// TIA Portal project "test项目" (V20)

(* hardware
DEVICE "S7-1200 station_1"  S7-1200 Station
   slot 0: "Rack_0"  S7-1200 Rack  Rack  V1.0
   slot 1: "PLC_1"  CPU 1215C DC/DC/DC  6ES7 215-1AG40-0XB0  V4.6
   slot 3: "CB 1241 (RS485)"  CB 1241 (RS485)  6ES7 241-1CH30-1XB0  V1.0
*)

// ===== PLC "PLC_1"  CPU 1215C DC/DC/DC =====

VAR_GLOBAL   // PLC tag table "默认变量表"
   "System_Byte" AT %MB1 : Byte;
   "FirstScan" AT %M1.0 : Bool;
   "DiagStatusUpdate" AT %M1.1 : Bool;
   "AlwaysTRUE" AT %M1.2 : Bool;
   "AlwaysFALSE" AT %M1.3 : Bool;
   "Clock_Byte" AT %MB0 : Byte;
   "Clock_10Hz" AT %M0.0 : Bool;
   "Clock_5Hz" AT %M0.1 : Bool;
   "Clock_2.5Hz" AT %M0.2 : Bool;
   "Clock_2Hz" AT %M0.3 : Bool;
   "Clock_1.25Hz" AT %M0.4 : Bool;
   "Clock_1Hz" AT %M0.5 : Bool;
   "Clock_0.625Hz" AT %M0.6 : Bool;
   "Clock_0.5Hz" AT %M0.7 : Bool;
   "Tag_1" AT %Q0.6 : Bool;
   "Tag_2" AT %I0.3 : Bool;
   "Tag_3" AT %I0.4 : Bool;
   "Tag_4" AT %I0.5 : Bool;
   "Tag_5" AT %I0.6 : Bool;
   "Tag_6" AT %I0.7 : Bool;
   "Tag_7" AT %M2.4 : Bool;
   "Tag_8" AT %M2.5 : Bool;
   "Tag_9" AT %M2.3 : Bool;
   "Tag_10" AT %QB0 : Byte;
END_VAR

VAR_GLOBAL   // PLC tag table "input"
   "limit_left" AT %I0.0 : Bool;
   "zero_point" AT %I0.1 : Bool;
   "limit_right" AT %I0.2 : Bool;
   "start" AT %I0.0 : Bool;
   "reset" AT %I0.1 : Bool;
   "b_a" AT %I0.2 : Bool;
   "b_b" AT %I0.3 : Bool;
   "b_c" AT %I0.4 : Bool;
   "b_d" AT %I0.5 : Bool;
END_VAR

VAR_GLOBAL   // PLC tag table "output"
   "puls_plus" AT %Q0.0 : Bool;
   "red_w" AT %Q0.1 : Bool;
   "dir_plus" AT %Q0.2 : Bool;
   "light_a" AT %Q0.3 : Bool;
   "light_b" AT %Q0.4 : Bool;
   "light_c" AT %Q0.5 : Bool;
   "light_d" AT %Q0.6 : Bool;
   "light_answer" AT %Q0.7 : Bool;
   "sound_answer" AT %Q1.2 : Bool;
END_VAR

VAR_GLOBAL   // PLC tag table "intermedia"
   "p1" AT %M2.0 : Bool;
   "p2" AT %M2.1 : Bool;
END_VAR

DATA_BLOCK "抢答器FB_SCL_DB"   // DB6
{ S7_Optimized_Access := 'TRUE' }
VERSION : 0.1
// stored: InstanceOfName 抢答器FB_SCL
"抢答器FB_SCL"
BEGIN
END_DATA_BLOCK

// folder: 作业

DATA_BLOCK "喷泉LAD数据块"   // DB1
{ S7_Optimized_Access := 'TRUE' }
VERSION : 0.1
   VAR
      started : Bool;
      stopped : Bool;
      running : Bool;
      cache : Array[0..10] of Bool;
      step1 : USInt;
      step2 : USInt;
      Static_1 : USInt;
      timer1 : IEC_TIMER;
      timer2 : IEC_TIMER;
      timer3 : IEC_TIMER;
      timer4 : IEC_TIMER;
      timer5 : IEC_TIMER;
      timer6 : IEC_TIMER;
      timer7 : IEC_TIMER;
      timer8 : IEC_TIMER;
      timer9 : IEC_TIMER;
      timer10 : IEC_TIMER;
      pt_1 : Time;
      pt_2 : Time;
   END_VAR
BEGIN
END_DATA_BLOCK

DATA_BLOCK "交通红绿灯_流程SCL_DB"   // DB2
{ S7_Optimized_Access := 'TRUE' }
VERSION : 0.1
// stored: InstanceOfName 交通红绿灯_流程SCL
"交通红绿灯_流程SCL"
BEGIN
END_DATA_BLOCK

DATA_BLOCK "交通红绿灯_比较SCL_DB"   // DB3
{ S7_Optimized_Access := 'TRUE' }
VERSION : 0.1
// stored: InstanceOfName 交通红绿灯_比较SCL
"交通红绿灯_比较SCL"
BEGIN
END_DATA_BLOCK

DATA_BLOCK "喷泉_DB"   // DB4
{ S7_Optimized_Access := 'TRUE' }
VERSION : 0.1
// stored: InstanceOfName 喷泉
"喷泉"
BEGIN
END_DATA_BLOCK

DATA_BLOCK "抢答器LAD数据块_1"   // DB5
{ S7_Optimized_Access := 'TRUE' }
VERSION : 0.1
   VAR
      started : Bool;
      success : Bool;
      success_a : Bool;
      success_b : Bool;
      success_c : Bool;
      success_d : Bool;
      cache : Array[0..10] of Bool;
      timer1 : IEC_TIMER;
      timer2 : IEC_TIMER;
      timer3 : IEC_TIMER;
      timer8 : IEC_TIMER;
      timer9 : IEC_TIMER;
      timer7 : IEC_TIMER;
      timer6 : IEC_TIMER;
      timer5 : IEC_TIMER;
      timer4 : IEC_TIMER;
      eligible_a : Bool;
      eligible_b : Bool;
      eligible_c : Bool;
      eligible_d : Bool;
      cnt : SInt;
   END_VAR
BEGIN
END_DATA_BLOCK

// folder: (top level)

FUNCTION_BLOCK "抢答器FB_SCL"   // FB4, SCL
{ S7_Optimized_Access := 'TRUE' }
VERSION : 0.1
   VAR
      started : Bool;
      start_TRIG_Instance : R_TRIG;
      reset_TRIG_Instance : R_TRIG;
      b_a_TRIG_Instance : R_TRIG;
      b_b_TRIG_Instance : R_TRIG;
      b_c_TRIG_Instance : R_TRIG;
      b_d_TRIG_Instance : R_TRIG;
      success_a : Bool;
      success_b : Bool;
      success_c : Bool;
      success_d : Bool;
      eligible_a : Bool;
      eligible_b : Bool;
      eligible_c : Bool;
      eligible_d : Bool;
      timer1 : IEC_TIMER;
      timer2 : IEC_TIMER;
      IEC_Timer_0_Instance : TON_TIME;
      IEC_Timer_0_Instance_1 : TON_TIME;
      IEC_Timer_0_Instance_2 : TON_TIME;
      pt_1 : Time;
      pt_2 : Time;
      pt_3 : Time;
      cnt : SInt;
   END_VAR
BEGIN
   If "FirstScan" THEN
       #started := 0;
   END_IF;

   #start_TRIG_Instance(CLK := "start");
   #reset_TRIG_Instance(CLK := "reset");
   #b_a_TRIG_Instance(CLK := "b_a");
   #b_b_TRIG_Instance(CLK := "b_b");
   #b_c_TRIG_Instance(CLK := "b_c");
   #b_d_TRIG_Instance(CLK := "b_d");
   #pt_1 := t#3s;
   #pt_2 := #pt_3 := t#1s;
   #IEC_Timer_0_Instance(IN := #started,
                         PT := #pt_1);

   #IEC_Timer_0_Instance_1(IN := #IEC_Timer_0_Instance.Q,
                           PT := #pt_2);

   #IEC_Timer_0_Instance_2(IN := #IEC_Timer_0_Instance_1.Q,
                           PT := #pt_3);

   If #start_TRIG_Instance.Q AND NOT #started THEN
       #started := #eligible_a := #eligible_b := #eligible_c := #eligible_d := 1;
       #success_a := #success_b := #success_c := #success_d := 0;
       #cnt := 0;

   END_IF;

   If #reset_TRIG_Instance.Q THEN
       #started := 0;
       "light_a" := "light_b" := "light_c" := "light_d" := "light_answer" := "sound_answer" := 0;
   END_IF;

   If #started THEN
       If NOT #IEC_Timer_0_Instance.Q THEN
           "light_a" := #eligible_a;
           "light_b" := #eligible_b;
           "light_c" := #eligible_c;
           "light_d" := #eligible_d;
           "light_answer" := "sound_answer" := 1;
           If #b_a_TRIG_Instance.Q THEN
               #eligible_a := 0;
           END_IF;
           If #b_b_TRIG_Instance.Q THEN
               #eligible_b := 0;
           END_IF;
           If #b_c_TRIG_Instance.Q THEN
               #eligible_c := 0;
           END_IF;
           If #b_d_TRIG_Instance.Q THEN
               #eligible_d := 0;
           END_IF;
       END_IF;

       If #IEC_Timer_0_Instance.Q THEN
           "light_a" := "light_b" := "light_c" := "light_d" := 0;
           If #eligible_a AND #b_a_TRIG_Instance.Q THEN
               #eligible_b := 0;
               #eligible_c := 0;
               #eligible_d := 0;
               #eligible_a := 0;
               #success_a := 1;
               RESET_TIMER(#IEC_Timer_0_Instance_1);
           END_IF;
           If #eligible_b AND #b_b_TRIG_Instance.Q THEN
               #eligible_b := 0;
               #eligible_c := 0;
               #eligible_d := 0;
               #eligible_a := 0;
               #success_b := 1;
               RESET_TIMER(#IEC_Timer_0_Instance_1);
           END_IF;
           If #eligible_c AND #b_c_TRIG_Instance.Q THEN
               #eligible_b := 0;
               #eligible_c := 0;
               #eligible_d := 0;
               #eligible_a := 0;
               #success_c := 1;
               RESET_TIMER(#IEC_Timer_0_Instance_1);
           END_IF;
           If #eligible_d AND #b_d_TRIG_Instance.Q THEN
               #eligible_b := 0;
               #eligible_c := 0;
               #eligible_d := 0;
               #eligible_a := 0;
               #success_d := 1;
               RESET_TIMER(#IEC_Timer_0_Instance_1);
           END_IF;

           If #success_a THEN
               "light_a" := NOT #IEC_Timer_0_Instance_1.Q OR #cnt = 3;
               If #IEC_Timer_0_Instance_2.Q THEN
                   RESET_TIMER(#IEC_Timer_0_Instance_1);
                   #cnt += 1;
               END_IF;
               If #cnt = 3 THEN
                   RESET_TIMER(#IEC_Timer_0_Instance_1);
               END_IF;
           END_IF;
           If #success_b THEN
               "light_b" := NOT #IEC_Timer_0_Instance_1.Q OR #cnt = 3;
               If #IEC_Timer_0_Instance_2.Q THEN
                   RESET_TIMER(#IEC_Timer_0_Instance_1);
                   #cnt += 1;
               END_IF;
               If #cnt = 3 THEN
                   RESET_TIMER(#IEC_Timer_0_Instance_1);
               END_IF;
           END_IF;
           If #success_c THEN
               "light_c" := NOT #IEC_Timer_0_Instance_1.Q OR #cnt = 3;
               If #IEC_Timer_0_Instance_2.Q THEN
                   RESET_TIMER(#IEC_Timer_0_Instance_1);
                   #cnt += 1;
               END_IF;
               If #cnt = 3 THEN
                   RESET_TIMER(#IEC_Timer_0_Instance_1);
               END_IF;
           END_IF;
           If #success_d THEN
               "light_d" := NOT #IEC_Timer_0_Instance_1.Q OR #cnt = 3;
               If #IEC_Timer_0_Instance_2.Q THEN
                   RESET_TIMER(#IEC_Timer_0_Instance_1);
                   #cnt += 1;
               END_IF;
               If #cnt = 3 THEN
                   RESET_TIMER(#IEC_Timer_0_Instance_1);
               END_IF;
           END_IF;
       END_IF;
   END_IF;
END_FUNCTION_BLOCK

ORGANIZATION_BLOCK "Main"   // OB1, LAD, ProgramCycle
TITLE = "Main Program Sweep (Cycle)"
{ S7_Optimized_Access := 'TRUE' }
VERSION : 0.1
   VAR_INPUT
      Initial_Call : Bool;   // Initial call of this OB
      Remanence : Bool;   // =True, if remanent data are available
   END_VAR
BEGIN

REGION Network 1 (SCL)
   (*



   *)
END_REGION

REGION Network 2
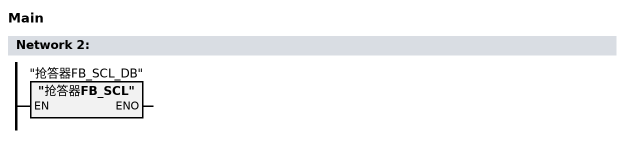
   RUNG wire#powerrail
      "抢答器FB_SCL_DB"()
   END_RUNG
   // the same network as SCL:
   "抢答器FB_SCL_DB"();   // "抢答器FB_SCL"
END_REGION
END_ORGANIZATION_BLOCK

// folder: 作业

FUNCTION_BLOCK "喷泉"   // FB1, SCL
{ S7_Optimized_Access := 'TRUE' }
VERSION : 0.1
   VAR
      timer1 : TON_TIME;
      timer2 : TON_TIME;
      pt_1 : Time;
      pt_2 : Time;
      step1 : USInt;
      step2 : USInt;
      step3 : USInt;
      started : Bool;
      stopped : Bool;
      running : Bool;
      R_TRIG_Instance : R_TRIG;
      R_TRIG_Instance_1 : R_TRIG;
      R_TRIG_Instance_2 : R_TRIG;
   END_VAR
BEGIN
   #timer1(IN := #running,
           PT := #pt_1);
   #timer2(IN := #timer1.Q,
           PT := #pt_2);
   #R_TRIG_Instance(CLK:="start");
   #R_TRIG_Instance_1(CLK:="reset");
   #R_TRIG_Instance_2(CLK:=#started);

   IF #R_TRIG_Instance.Q THEN
       #started := 1;
   END_IF;

   IF #R_TRIG_Instance_1.Q THEN
       #stopped := 1;
   END_IF;

   IF #R_TRIG_Instance_2.Q THEN
       #running := 1;
       #pt_1 := t#5s;
       #pt_2 := t#5s;
       RESET_TIMER(#timer1);
       #step1 := #step2 := #step3 := 0;
   END_IF;

   IF #running THEN
       IF #step1 = 0 THEN
           "light_a" := NOT #timer1.Q;
           "light_b" := NOT #timer2.Q AND #timer1.Q;
           IF #timer2.Q THEN
               #step1 += 1;
               RESET_TIMER(#timer1);
           END_IF;
       END_IF;

       IF #step1 = 1 THEN
           "light_a" := "light_b" := NOT #timer1.Q;
           IF #timer1.Q THEN
               #step1 += 1;
               #pt_1 := #pt_2 := t#1s;
               RESET_TIMER(#timer1);
           END_IF;
       END_IF;

       IF #step1 = 2 THEN
           "light_c" := NOT #timer1.Q;
           IF #timer2.Q THEN
               #step2 += 1;
               RESET_TIMER(#timer1);
           END_IF;
           IF #step2 = 5 THEN
               #step1 += 1;
               #pt_1 := t#5s;
               RESET_TIMER(#timer1);
               #step2 := 0;
           END_IF;
       END_IF;

       IF #step1 = 3 THEN
           "light_a" := "light_b" := NOT #timer1.Q;
           IF #timer1.Q THEN
               #step1 += 1;
               #pt_1 := t#2s;
               RESET_TIMER(#timer1);
           END_IF;
       END_IF;

       IF #step1 = 4 THEN
           CASE #step3 OF
               0:
                   "light_a" := NOT #timer1.Q;
               1:
                   "light_b" := NOT #timer1.Q;
               2:
                   "light_c" := NOT #timer1.Q;
           END_CASE;

           IF #timer1.Q THEN
               #step3 += 1;
               IF #step3 = 3 THEN
                   #step2 += 1;
                   #step3 := 0;
               END_IF;
               IF #step2 = 3 THEN
                   #step1 += 1;
                   #step2 := 0;
                   #pt_1 := t#5S;
               END_IF;
               RESET_TIMER(#timer1);
           END_IF;
       END_IF;

       IF #step1 = 5 THEN
           IF #timer1.Q THEN
               #running := NOT #stopped;
               #started := #running;
               #pt_1 := #pt_2 := t#5s;
               #step1 := #step2 := #step3 := 0;
               RESET_TIMER(#timer1);
           END_IF;
       END_IF;
   END_IF;
END_FUNCTION_BLOCK

FUNCTION_BLOCK "交通红绿灯_流程SCL"   // FB2, LAD
{ S7_Optimized_Access := 'TRUE' }
VERSION : 0.1
   VAR
      start_pressed_trig : R_TRIG;
      stop_pressed_trig : R_TRIG;
      start_trig : R_TRIG;
      started : Bool;
      stoped : Bool;
      step_w : Byte;
      step_s : Byte;
      Timer_0 : TON_TIME;
      Timer_1 : TON_TIME;
      Timer_2 : TON_TIME;
      Timer_3 : TON_TIME;
      time_w : Time;
      time_s : Time;
   END_VAR
BEGIN

REGION Network 2 (SCL)
   IF "FirstScan" THEN
       #started := #stoped := 0;
       #step_w := #step_s := 0;
   END_IF;

   //initiate
   #start_pressed_trig(CLK := "limit_left");
   #stop_pressed_trig(CLK := "zero_point");
   #start_trig(CLK := #started);

   #Timer_0(IN := #started, PT := #time_w);
   #Timer_1(IN := #started, PT := #time_s);
   #Timer_2(IN := "AlwaysTRUE", PT := t#500ms);
   #Timer_3(IN := #Timer_2.Q,PT := t#500ms);
   IF #Timer_3.Q THEN
       RESET_TIMER(#Timer_2);
   END_IF;

   IF #start_pressed_trig.Q THEN
       #started := 1;
       #stoped := 0;
   END_IF;

   IF #start_trig.Q THEN
       #stoped := 0;
       #step_s := #step_w := 0;
       "light_a" := "puls_plus" := "dir_plus" := "light_c" := "red_w" := "light_b" := 0;
       #time_w := t#5s;
       #time_s := t#10s;
       RESET_TIMER(#Timer_0);
       RESET_TIMER(#Timer_1);
   END_IF;

   IF #stop_pressed_trig.Q THEN
       #stoped := 1;
   END_IF;

   IF #started THEN
       //东西向
       IF #step_w = 0 THEN
           "puls_plus" := 1;
           IF #Timer_0.Q THEN
               "puls_plus" := 0;
               RESET_TIMER(#Timer_0);
               #time_w := T#3s;
               #step_w += 1;
           END_IF;
       END_IF;

       IF #step_w = 1 THEN
           "puls_plus" := #Timer_2.Q;
           IF #Timer_0.Q THEN
               "puls_plus" := 0;
               RESET_TIMER(#Timer_0);
               #time_w := T#2s;
               #step_w += 1;
           END_IF;
       END_IF;

       IF #step_w = 2 THEN
           "dir_plus" := 1;
           IF #Timer_0.Q THEN
               "dir_plus" := 0;
               RESET_TIMER(#Timer_0);
               #time_w := T#10s;
               #step_w += 1;
           END_IF;
       END_IF;

       IF #step_w = 3 THEN
           "red_w":= 1;
           IF #Timer_0.Q THEN
               "red_w" := 0;
               RESET_TIMER(#Timer_0);
               #time_w := T#5s;
               #step_w := 0;
           END_IF;
       END_IF;

       //南北向
       IF #step_s = 0 THEN
           "light_b" := 1;
           IF #Timer_1.Q THEN
               "light_b" := 0;
               RESET_TIMER(#Timer_1);
               #time_s := T#5s;
               #step_s += 1;
           END_IF;
       END_IF;

       IF #step_s = 1 THEN
           "light_a" := 1;
           IF #Timer_1.Q THEN
               "light_a" := 0;
               RESET_TIMER(#Timer_1);
               #time_s := T#3s;
               #step_s += 1;
           END_IF;
       END_IF;

       IF #step_s = 2 THEN
          "light_a" := #Timer_2.Q;
          IF #Timer_1.Q THEN
              "light_a" := 0;
               RESET_TIMER(#Timer_1);
               #time_s := T#2s;
               #step_s += 1;
           END_IF;
       END_IF;

       IF #step_s = 3 THEN
           "light_c" := 1;
           IF #Timer_1.Q THEN
               "light_c" := 0;
               RESET_TIMER(#Timer_1);
               #time_s := T#10s;
               #step_s := 0;
               #step_w := 0;
               "red_w" := 0;
               RESET_TIMER(#Timer_0);
               #time_w := T#5s;
               #step_w := 0;

               IF #stoped THEN
                   #started := 0;
                   #stoped := 0;
               END_IF;
           END_IF;
       END_IF;
   END_IF;

   IF NOT #stoped AND NOT #started THEN
       "light_c" := #Timer_2.Q;
       "dir_plus" := #Timer_2.Q;
   END_IF;
END_REGION
END_FUNCTION_BLOCK

FUNCTION_BLOCK "交通红绿灯_比较SCL"   // FB3, LAD
{ S7_Optimized_Access := 'TRUE' }
VERSION : 0.1
   VAR
      start_pressed_trig : R_TRIG;
      stop_pressed_trig : R_TRIG;
      start_trig : R_TRIG;
      started : Bool;
      stoped : Bool;
      step_w : Byte;
      step_s : Byte;
      Timer_0 : TON_TIME;
      Timer_1 : TON_TIME;
      Timer_2 : TON_TIME;
      Timer_3 : TON_TIME;
      time_w : Time;
      time_s : Time;
      button : Array[0..10] of Bool;
      b1 : Bool;
      b2 : Bool;
      b4 : Bool;
      b3 : Bool;
      b5 : Bool;
   END_VAR
BEGIN

REGION Network 2 (SCL)
   IF "FirstScan" THEN
       #started := #stoped := 0;
       #step_w := #step_s := 0;
   END_IF;

   //initiate
   #start_pressed_trig(CLK := "limit_left");
   #stop_pressed_trig(CLK := "zero_point");
   #start_trig(CLK := #started);

   #Timer_0(IN := #started, PT := t#20S);
   #Timer_2(IN := "AlwaysTRUE", PT := t#500ms);
   #Timer_3(IN := #Timer_2.Q,PT := t#500ms);
   IF #Timer_3.Q THEN
       RESET_TIMER(#Timer_2);
   END_IF;

   IF #start_pressed_trig.Q THEN
       #started := 1;
       #stoped := 0;
   END_IF;

   IF #start_trig.Q THEN
       #stoped := 0;
       RESET_TIMER(#Timer_0);
       RESET_TIMER(#Timer_2);
   END_IF;

   IF #stop_pressed_trig.Q THEN
       #stoped := 1;
   END_IF;

   IF #started THEN
       //东西向
       "puls_plus" := #Timer_0.ET > t#0s AND #Timer_0.ET <= t#5s OR (#Timer_0.ET > t#5s AND #Timer_0.ET <= t#8s AND #Timer_2.Q);
       "dir_plus" := #Timer_0.ET > t#8s AND #Timer_0.ET <= t#10s;
       "red_w" := #Timer_0.ET > t#10s AND #Timer_0.ET <= t#20s;

       //南北向
       "light_b" := #Timer_0.ET > t#0s AND #Timer_0.ET <= t#10s;
       "light_a" := #Timer_0.ET > t#10s AND #Timer_0.ET <= t#13s OR (#Timer_0.ET > t#13s AND #Timer_0.ET <= t#15s AND #Timer_2.Q);
       "light_c" := #Timer_0.ET > t#15s AND #Timer_0.ET < t#20s;

       IF #Timer_0.ET >= t#20S THEN
           RESET_TIMER(#Timer_0);
           RESET_TIMER(#Timer_1);

           #started := NOT #stoped;
           #stoped := 0;
       END_IF;
   END_IF;

   IF NOT #stoped AND NOT #started THEN
       "light_a" := "puls_plus" := "light_b" := "red_w" := 0;
       "light_c" := #Timer_2.Q;
       "dir_plus" := #Timer_2.Q;
   END_IF;
END_REGION
END_FUNCTION_BLOCK

FUNCTION "红绿灯_FC" : Void   // FC1, LAD
{ S7_Optimized_Access := 'TRUE' }
VERSION : 0.1
   VAR_TEMP   // added for the SCL form of the ladder/FBD networks
      _w1 : Bool;
      _w2 : Bool;
      _w3 : Bool;
   END_VAR
BEGIN

REGION Network 1
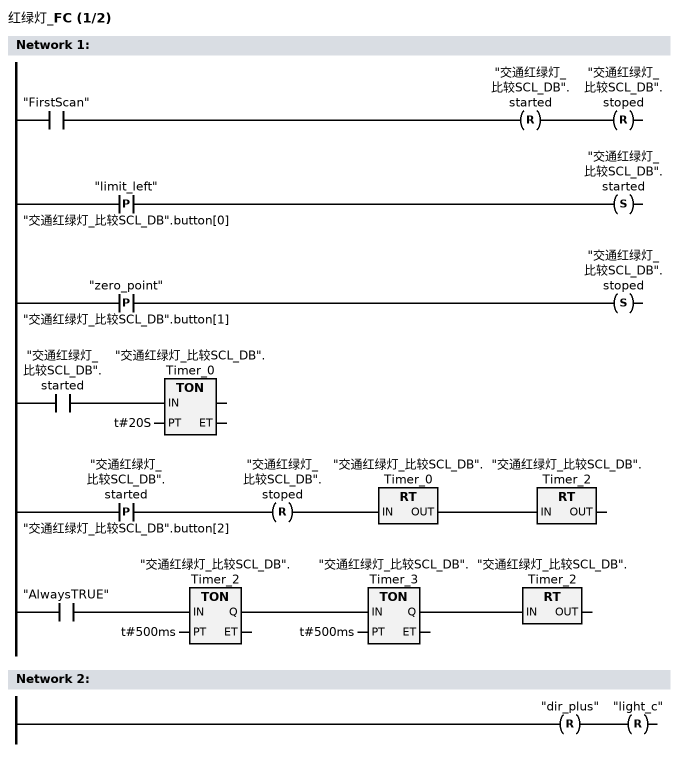
   IF "FirstScan" THEN
       "交通红绿灯_比较SCL_DB".started := FALSE;
       "交通红绿灯_比较SCL_DB".stoped := FALSE;
   END_IF;
   #_w1 := "limit_left" AND NOT "交通红绿灯_比较SCL_DB".button[0];   // rising edge of "limit_left"
   "交通红绿灯_比较SCL_DB".button[0] := "limit_left";
   IF #_w1 THEN "交通红绿灯_比较SCL_DB".started := TRUE; END_IF;
   #_w2 := "zero_point" AND NOT "交通红绿灯_比较SCL_DB".button[1];   // rising edge of "zero_point"
   "交通红绿灯_比较SCL_DB".button[1] := "zero_point";
   IF #_w2 THEN "交通红绿灯_比较SCL_DB".stoped := TRUE; END_IF;
   "交通红绿灯_比较SCL_DB".Timer_0.TON(IN := "交通红绿灯_比较SCL_DB".started, PT := t#20S);
   #_w3 := "交通红绿灯_比较SCL_DB".started AND NOT "交通红绿灯_比较SCL_DB".button[2];   // rising edge of "交通红绿灯_比较SCL_DB".started
   "交通红绿灯_比较SCL_DB".button[2] := "交通红绿灯_比较SCL_DB".started;
   IF #_w3 THEN
       "交通红绿灯_比较SCL_DB".stoped := FALSE;
       RESET_TIMER("交通红绿灯_比较SCL_DB".Timer_0);
       RESET_TIMER("交通红绿灯_比较SCL_DB".Timer_2);
   END_IF;
   "交通红绿灯_比较SCL_DB".Timer_2.TON(IN := "AlwaysTRUE", PT := t#500ms);
   "交通红绿灯_比较SCL_DB".Timer_3.TON(IN := "交通红绿灯_比较SCL_DB".Timer_2.Q, PT := t#500ms);
   IF "交通红绿灯_比较SCL_DB".Timer_3.Q THEN RESET_TIMER("交通红绿灯_比较SCL_DB".Timer_2); END_IF;
END_REGION

REGION Network 2
   RUNG wire#powerrail
      R_Coil( "dir_plus" )
      R_Coil( "light_c" )
   END_RUNG
   // the same network as SCL:
   "dir_plus" := FALSE;
   "light_c" := FALSE;
END_REGION

REGION Network 3
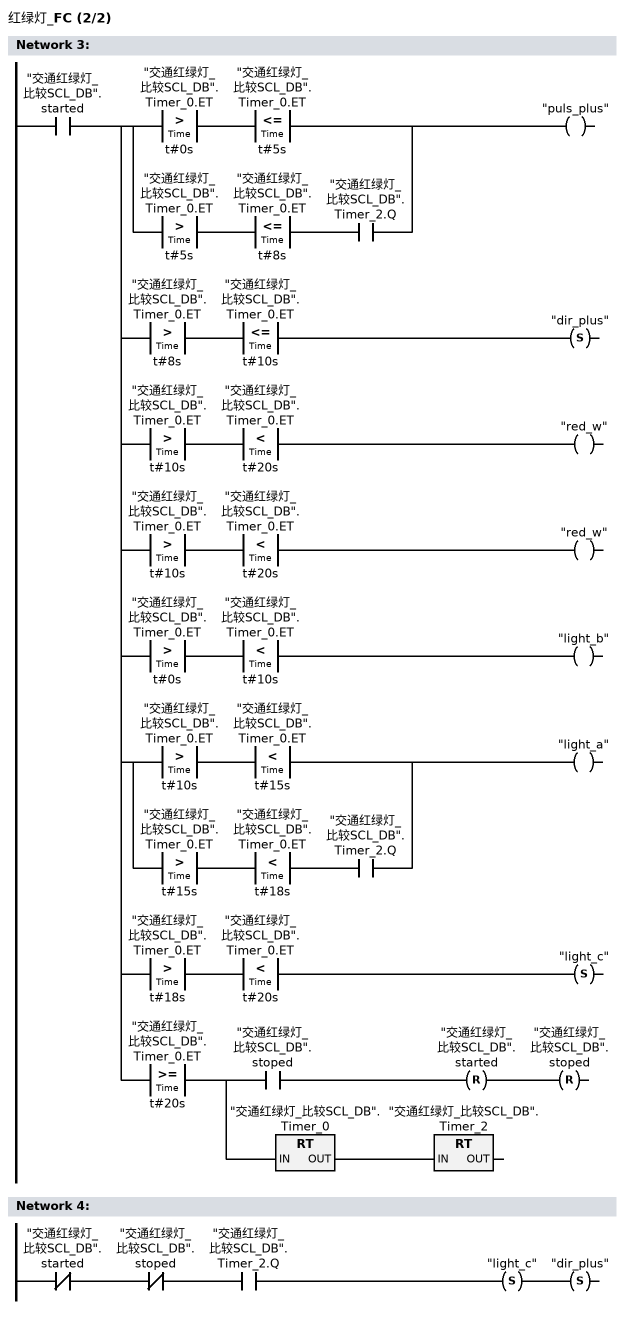
   RUNG wire#powerrail
      Contact( "交通红绿灯_比较SCL_DB".started )
      wire#w1
      { S7_Templates := "SrcType := Time" } GT_Contact(in1 := "交通红绿灯_比较SCL_DB".Timer_0.ET, in2 := t#0s)
      { S7_Templates := "SrcType := Time" } LE_Contact(in1 := "交通红绿灯_比较SCL_DB".Timer_0.ET, in2 := t#5s)
      wire#w2
      Coil( "puls_plus" )
   END_RUNG
   RUNG wire#w1
      { S7_Templates := "SrcType := Time" } GT_Contact(in1 := "交通红绿灯_比较SCL_DB".Timer_0.ET, in2 := t#5s)
      { S7_Templates := "SrcType := Time" } LE_Contact(in1 := "交通红绿灯_比较SCL_DB".Timer_0.ET, in2 := t#8s)
      Contact( "交通红绿灯_比较SCL_DB".Timer_2.Q )
   END_RUNG wire#w2
   RUNG wire#w1
      { S7_Templates := "SrcType := Time" } GT_Contact(in1 := "交通红绿灯_比较SCL_DB".Timer_0.ET, in2 := t#8s)
      { S7_Templates := "SrcType := Time" } LE_Contact(in1 := "交通红绿灯_比较SCL_DB".Timer_0.ET, in2 := t#10s)
      S_Coil( "dir_plus" )
   END_RUNG
   RUNG wire#w1
      { S7_Templates := "SrcType := Time" } GT_Contact(in1 := "交通红绿灯_比较SCL_DB".Timer_0.ET, in2 := t#10s)
      { S7_Templates := "SrcType := Time" } LT_Contact(in1 := "交通红绿灯_比较SCL_DB".Timer_0.ET, in2 := t#20s)
      Coil( "red_w" )
   END_RUNG
   RUNG wire#w1
      { S7_Templates := "SrcType := Time" } GT_Contact(in1 := "交通红绿灯_比较SCL_DB".Timer_0.ET, in2 := t#10s)
      { S7_Templates := "SrcType := Time" } LT_Contact(in1 := "交通红绿灯_比较SCL_DB".Timer_0.ET, in2 := t#20s)
      Coil( "red_w" )
   END_RUNG
   RUNG wire#w1
      { S7_Templates := "SrcType := Time" } GT_Contact(in1 := "交通红绿灯_比较SCL_DB".Timer_0.ET, in2 := t#0s)
      { S7_Templates := "SrcType := Time" } LT_Contact(in1 := "交通红绿灯_比较SCL_DB".Timer_0.ET, in2 := t#10s)
      Coil( "light_b" )
   END_RUNG
   RUNG wire#w1
      { S7_Templates := "SrcType := Time" } GT_Contact(in1 := "交通红绿灯_比较SCL_DB".Timer_0.ET, in2 := t#10s)
      { S7_Templates := "SrcType := Time" } LT_Contact(in1 := "交通红绿灯_比较SCL_DB".Timer_0.ET, in2 := t#15s)
      wire#w3
      Coil( "light_a" )
   END_RUNG
   RUNG wire#w1
      { S7_Templates := "SrcType := Time" } GT_Contact(in1 := "交通红绿灯_比较SCL_DB".Timer_0.ET, in2 := t#15s)
      { S7_Templates := "SrcType := Time" } LT_Contact(in1 := "交通红绿灯_比较SCL_DB".Timer_0.ET, in2 := t#18s)
      Contact( "交通红绿灯_比较SCL_DB".Timer_2.Q )
   END_RUNG wire#w3
   RUNG wire#w1
      { S7_Templates := "SrcType := Time" } GT_Contact(in1 := "交通红绿灯_比较SCL_DB".Timer_0.ET, in2 := t#18s)
      { S7_Templates := "SrcType := Time" } LT_Contact(in1 := "交通红绿灯_比较SCL_DB".Timer_0.ET, in2 := t#20s)
      S_Coil( "light_c" )
   END_RUNG
   RUNG wire#w1
      { S7_Templates := "SrcType := Time" } GE_Contact(in1 := "交通红绿灯_比较SCL_DB".Timer_0.ET, in2 := t#20s)
      wire#w4
      Contact( "交通红绿灯_比较SCL_DB".stoped )
      R_Coil( "交通红绿灯_比较SCL_DB".started )
      R_Coil( "交通红绿灯_比较SCL_DB".stoped )
   END_RUNG
   RUNG wire#w4
      RT_Coil( "交通红绿灯_比较SCL_DB".Timer_0 )
      RT_Coil( "交通红绿灯_比较SCL_DB".Timer_2 )
   END_RUNG
   // the same network as SCL:
   "puls_plus" := "交通红绿灯_比较SCL_DB".started AND ((("交通红绿灯_比较SCL_DB".Timer_0.ET > t#0s) AND ("交通红绿灯_比较SCL_DB".Timer_0.ET <= t#5s)) OR (("交通红绿灯_比较SCL_DB".Timer_0.ET > t#5s) AND ("交通红绿灯_比较SCL_DB".Timer_0.ET <= t#8s) AND "交通红绿灯_比较SCL_DB".Timer_2.Q));
   IF "交通红绿灯_比较SCL_DB".started AND ("交通红绿灯_比较SCL_DB".Timer_0.ET > t#8s) AND ("交通红绿灯_比较SCL_DB".Timer_0.ET <= t#10s) THEN
       "dir_plus" := TRUE;
   END_IF;
   "red_w" := "交通红绿灯_比较SCL_DB".started AND ("交通红绿灯_比较SCL_DB".Timer_0.ET > t#10s) AND ("交通红绿灯_比较SCL_DB".Timer_0.ET < t#20s);
   "red_w" := "交通红绿灯_比较SCL_DB".started AND ("交通红绿灯_比较SCL_DB".Timer_0.ET > t#10s) AND ("交通红绿灯_比较SCL_DB".Timer_0.ET < t#20s);
   "light_b" := "交通红绿灯_比较SCL_DB".started AND ("交通红绿灯_比较SCL_DB".Timer_0.ET > t#0s) AND ("交通红绿灯_比较SCL_DB".Timer_0.ET < t#10s);
   "light_a" := "交通红绿灯_比较SCL_DB".started AND ((("交通红绿灯_比较SCL_DB".Timer_0.ET > t#10s) AND ("交通红绿灯_比较SCL_DB".Timer_0.ET < t#15s)) OR (("交通红绿灯_比较SCL_DB".Timer_0.ET > t#15s) AND ("交通红绿灯_比较SCL_DB".Timer_0.ET < t#18s) AND "交通红绿灯_比较SCL_DB".Timer_2.Q));
   IF "交通红绿灯_比较SCL_DB".started AND ("交通红绿灯_比较SCL_DB".Timer_0.ET > t#18s) AND ("交通红绿灯_比较SCL_DB".Timer_0.ET < t#20s) THEN
       "light_c" := TRUE;
   END_IF;
   #_w1 := "交通红绿灯_比较SCL_DB".started AND ("交通红绿灯_比较SCL_DB".Timer_0.ET >= t#20s);
   IF #_w1 AND "交通红绿灯_比较SCL_DB".stoped THEN
       "交通红绿灯_比较SCL_DB".started := FALSE;
       "交通红绿灯_比较SCL_DB".stoped := FALSE;
   END_IF;
   IF #_w1 THEN
       RESET_TIMER("交通红绿灯_比较SCL_DB".Timer_0);
       RESET_TIMER("交通红绿灯_比较SCL_DB".Timer_2);
   END_IF;
END_REGION

REGION Network 4
   RUNG wire#powerrail
      I_Contact( "交通红绿灯_比较SCL_DB".started )
      I_Contact( "交通红绿灯_比较SCL_DB".stoped )
      Contact( "交通红绿灯_比较SCL_DB".Timer_2.Q )
      S_Coil( "light_c" )
      S_Coil( "dir_plus" )
   END_RUNG
   // the same network as SCL:
   IF NOT "交通红绿灯_比较SCL_DB".started AND NOT "交通红绿灯_比较SCL_DB".stoped AND "交通红绿灯_比较SCL_DB".Timer_2.Q THEN
       "light_c" := TRUE;
       "dir_plus" := TRUE;
   END_IF;
END_REGION
END_FUNCTION

FUNCTION "喷泉作业" : Void   // FC2, LAD
{ S7_Optimized_Access := 'TRUE' }
VERSION : 0.1
   VAR_TEMP   // added for the SCL form of the ladder/FBD networks
      _w1 : Bool;
      _w2 : Bool;
      _w3 : Bool;
      _w4 : Bool;
      _w5 : Bool;
      _w6 : Bool;
      _w7 : Bool;
      _w8 : Bool;
      _w9 : Bool;
      _w10 : Bool;
      _w11 : Bool;
      _w12 : Bool;
   END_VAR
BEGIN

REGION Network 1
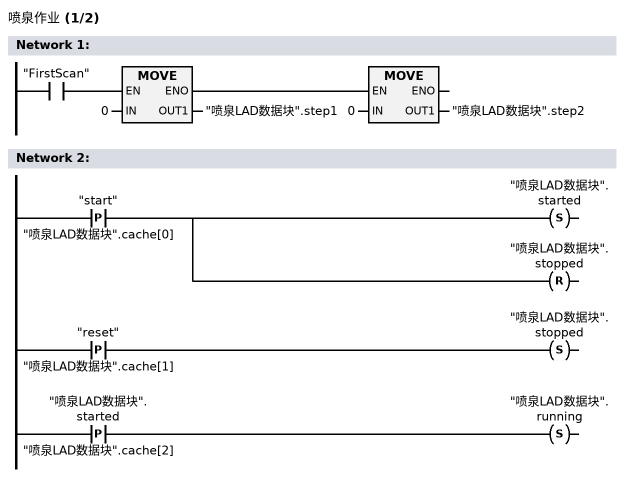
   RUNG wire#powerrail
      Contact( "FirstScan" )
      Move(in := 0, out1 => "喷泉LAD数据块".step1)
      Move(in := 0, out1 => "喷泉LAD数据块".step2)
   END_RUNG
   // the same network as SCL:
   IF "FirstScan" THEN
       "喷泉LAD数据块".step1 := 0;
       "喷泉LAD数据块".step2 := 0;
   END_IF;
END_REGION

REGION Network 2
   RUNG wire#powerrail
      P_Contact(operand := "start", bit := "喷泉LAD数据块".cache[0])
      wire#w1
      S_Coil( "喷泉LAD数据块".started )
   END_RUNG
   RUNG wire#w1
      R_Coil( "喷泉LAD数据块".stopped )
   END_RUNG
   RUNG wire#powerrail
      P_Contact(operand := "reset", bit := "喷泉LAD数据块".cache[1])
      S_Coil( "喷泉LAD数据块".stopped )
   END_RUNG
   RUNG wire#powerrail
      P_Contact(operand := "喷泉LAD数据块".started, bit := "喷泉LAD数据块".cache[2])
      S_Coil( "喷泉LAD数据块".running )
   END_RUNG
   // the same network as SCL:
   #_w1 := "start" AND NOT "喷泉LAD数据块".cache[0];   // rising edge of "start"
   "喷泉LAD数据块".cache[0] := "start";
   IF #_w1 THEN
       "喷泉LAD数据块".started := TRUE;
       "喷泉LAD数据块".stopped := FALSE;
   END_IF;
   #_w2 := "reset" AND NOT "喷泉LAD数据块".cache[1];   // rising edge of "reset"
   "喷泉LAD数据块".cache[1] := "reset";
   IF #_w2 THEN "喷泉LAD数据块".stopped := TRUE; END_IF;
   #_w3 := "喷泉LAD数据块".started AND NOT "喷泉LAD数据块".cache[2];   // rising edge of "喷泉LAD数据块".started
   "喷泉LAD数据块".cache[2] := "喷泉LAD数据块".started;
   IF #_w3 THEN "喷泉LAD数据块".running := TRUE; END_IF;
END_REGION

REGION Network 3
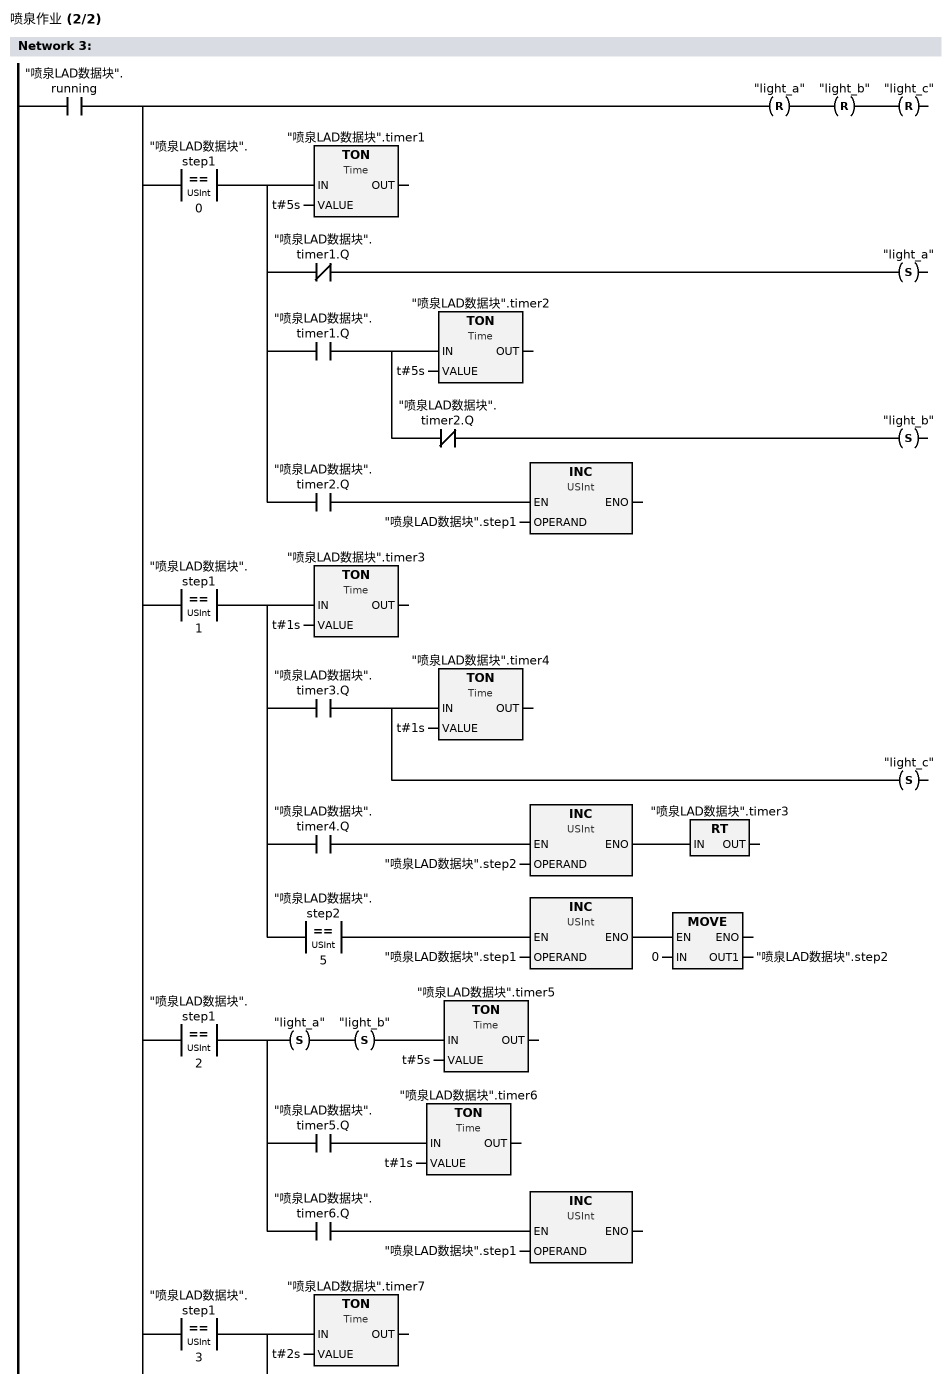
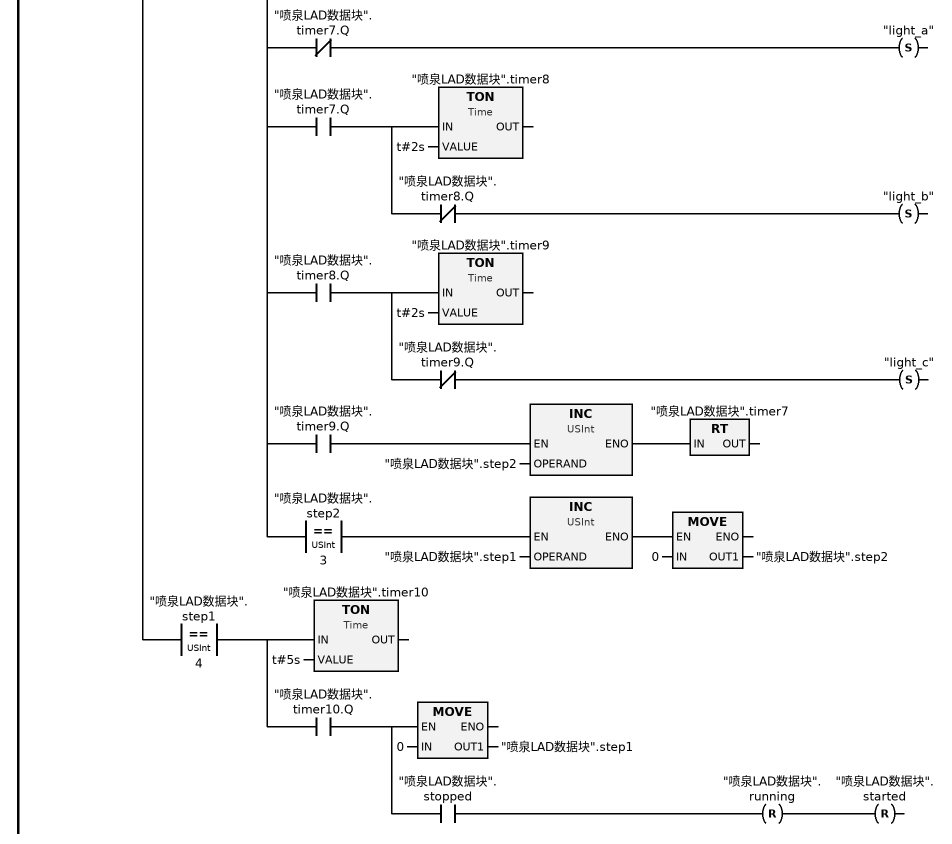
   IF "喷泉LAD数据块".running THEN
       "light_a" := FALSE;
       "light_b" := FALSE;
       "light_c" := FALSE;
   END_IF;
   #_w1 := "喷泉LAD数据块".running AND ("喷泉LAD数据块".step1 = 0);
   "喷泉LAD数据块".timer1.TON(IN := #_w1, PT := t#5s);   // TON coil
   IF #_w1 AND NOT "喷泉LAD数据块".timer1.Q THEN "light_a" := TRUE; END_IF;
   #_w2 := #_w1 AND "喷泉LAD数据块".timer1.Q;
   "喷泉LAD数据块".timer2.TON(IN := #_w2, PT := t#5s);   // TON coil
   IF #_w2 AND NOT "喷泉LAD数据块".timer2.Q THEN "light_b" := TRUE; END_IF;
   IF #_w1 AND "喷泉LAD数据块".timer2.Q THEN "喷泉LAD数据块".step1 := "喷泉LAD数据块".step1 + 1; END_IF;
   #_w3 := "喷泉LAD数据块".running AND ("喷泉LAD数据块".step1 = 1);
   "喷泉LAD数据块".timer3.TON(IN := #_w3, PT := t#1s);   // TON coil
   #_w4 := #_w3 AND "喷泉LAD数据块".timer3.Q;
   "喷泉LAD数据块".timer4.TON(IN := #_w4, PT := t#1s);   // TON coil
   IF #_w4 THEN "light_c" := TRUE; END_IF;
   #_w5 := #_w3 AND "喷泉LAD数据块".timer4.Q;
   IF #_w5 THEN
       "喷泉LAD数据块".step2 := "喷泉LAD数据块".step2 + 1;
       RESET_TIMER("喷泉LAD数据块".timer3);
   END_IF;
   IF #_w3 AND ("喷泉LAD数据块".step2 = 5) THEN
       "喷泉LAD数据块".step1 := "喷泉LAD数据块".step1 + 1;
       "喷泉LAD数据块".step2 := 0;
   END_IF;
   #_w6 := "喷泉LAD数据块".running AND ("喷泉LAD数据块".step1 = 2);
   IF #_w6 THEN
       "light_a" := TRUE;
       "light_b" := TRUE;
   END_IF;
   "喷泉LAD数据块".timer5.TON(IN := #_w6, PT := t#5s);   // TON coil
   "喷泉LAD数据块".timer6.TON(IN := #_w6 AND "喷泉LAD数据块".timer5.Q, PT := t#1s);   // TON coil
   IF #_w6 AND "喷泉LAD数据块".timer6.Q THEN "喷泉LAD数据块".step1 := "喷泉LAD数据块".step1 + 1; END_IF;
   #_w7 := "喷泉LAD数据块".running AND ("喷泉LAD数据块".step1 = 3);
   "喷泉LAD数据块".timer7.TON(IN := #_w7, PT := t#2s);   // TON coil
   IF #_w7 AND NOT "喷泉LAD数据块".timer7.Q THEN "light_a" := TRUE; END_IF;
   #_w8 := #_w7 AND "喷泉LAD数据块".timer7.Q;
   "喷泉LAD数据块".timer8.TON(IN := #_w8, PT := t#2s);   // TON coil
   IF #_w8 AND NOT "喷泉LAD数据块".timer8.Q THEN "light_b" := TRUE; END_IF;
   #_w9 := #_w7 AND "喷泉LAD数据块".timer8.Q;
   "喷泉LAD数据块".timer9.TON(IN := #_w9, PT := t#2s);   // TON coil
   IF #_w9 AND NOT "喷泉LAD数据块".timer9.Q THEN "light_c" := TRUE; END_IF;
   #_w10 := #_w7 AND "喷泉LAD数据块".timer9.Q;
   IF #_w10 THEN
       "喷泉LAD数据块".step2 := "喷泉LAD数据块".step2 + 1;
       RESET_TIMER("喷泉LAD数据块".timer7);
   END_IF;
   IF #_w7 AND ("喷泉LAD数据块".step2 = 3) THEN
       "喷泉LAD数据块".step1 := "喷泉LAD数据块".step1 + 1;
       "喷泉LAD数据块".step2 := 0;
   END_IF;
   #_w11 := "喷泉LAD数据块".running AND ("喷泉LAD数据块".step1 = 4);
   "喷泉LAD数据块".timer10.TON(IN := #_w11, PT := t#5s);   // TON coil
   #_w12 := #_w11 AND "喷泉LAD数据块".timer10.Q;
   IF #_w12 THEN "喷泉LAD数据块".step1 := 0; END_IF;
   IF #_w12 AND "喷泉LAD数据块".stopped THEN
       "喷泉LAD数据块".running := FALSE;
       "喷泉LAD数据块".started := FALSE;
   END_IF;
END_REGION
END_FUNCTION

FUNCTION "抢答器LAD" : Void   // FC3, LAD
{ S7_Optimized_Access := 'TRUE' }
VERSION : 0.1
   VAR_TEMP   // added for the SCL form of the ladder/FBD networks
      _w1 : Bool;
      _w2 : Bool;
      _w3 : Bool;
      _w4 : Bool;
      _w5 : Bool;
      _w6 : Bool;
      _w7 : Bool;
      _w8 : Bool;
      _w9 : Bool;
      _w10 : Bool;
      _w11 : Bool;
      _w12 : Bool;
      _w13 : Bool;
      _w14 : Bool;
      _w15 : Bool;
      _w16 : Bool;
      _w17 : Bool;
      _w18 : Bool;
      _w19 : Bool;
      _w20 : Bool;
      _w21 : Bool;
      _w22 : Bool;
      _w23 : Bool;
      _w24 : Bool;
      _w25 : Bool;
      _w26 : Bool;
   END_VAR
BEGIN

REGION Network 1
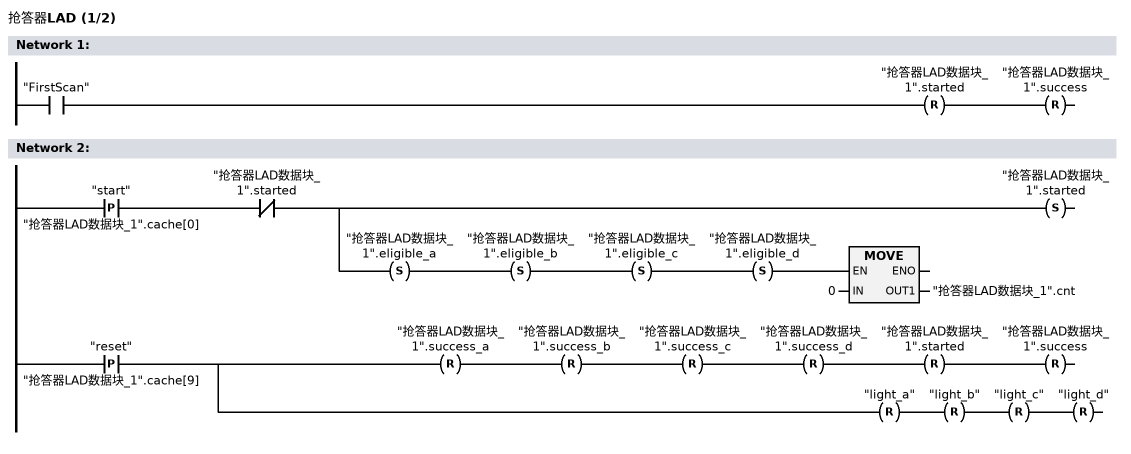
   RUNG wire#powerrail
      Contact( "FirstScan" )
      R_Coil( "抢答器LAD数据块_1".started )
      R_Coil( "抢答器LAD数据块_1".success )
   END_RUNG
   // the same network as SCL:
   IF "FirstScan" THEN
       "抢答器LAD数据块_1".started := FALSE;
       "抢答器LAD数据块_1".success := FALSE;
   END_IF;
END_REGION

REGION Network 2
   RUNG wire#powerrail
      P_Contact(operand := "start", bit := "抢答器LAD数据块_1".cache[0])
      I_Contact( "抢答器LAD数据块_1".started )
      wire#w1
      S_Coil( "抢答器LAD数据块_1".started )
   END_RUNG
   RUNG wire#w1
      S_Coil( "抢答器LAD数据块_1".eligible_a )
      S_Coil( "抢答器LAD数据块_1".eligible_b )
      S_Coil( "抢答器LAD数据块_1".eligible_c )
      S_Coil( "抢答器LAD数据块_1".eligible_d )
      Move(in := 0, out1 => "抢答器LAD数据块_1".cnt)
   END_RUNG
   RUNG wire#powerrail
      P_Contact(operand := "reset", bit := "抢答器LAD数据块_1".cache[9])
      wire#w2
      R_Coil( "抢答器LAD数据块_1".success_a )
      R_Coil( "抢答器LAD数据块_1".success_b )
      R_Coil( "抢答器LAD数据块_1".success_c )
      R_Coil( "抢答器LAD数据块_1".success_d )
      R_Coil( "抢答器LAD数据块_1".started )
      R_Coil( "抢答器LAD数据块_1".success )
   END_RUNG
   RUNG wire#w2
      R_Coil( "light_a" )
      R_Coil( "light_b" )
      R_Coil( "light_c" )
      R_Coil( "light_d" )
   END_RUNG
   // the same network as SCL:
   #_w1 := "start" AND NOT "抢答器LAD数据块_1".cache[0];   // rising edge of "start"
   "抢答器LAD数据块_1".cache[0] := "start";
   #_w2 := #_w1 AND NOT "抢答器LAD数据块_1".started;
   IF #_w2 THEN
       "抢答器LAD数据块_1".started := TRUE;
       "抢答器LAD数据块_1".eligible_a := TRUE;
       "抢答器LAD数据块_1".eligible_b := TRUE;
       "抢答器LAD数据块_1".eligible_c := TRUE;
       "抢答器LAD数据块_1".eligible_d := TRUE;
       "抢答器LAD数据块_1".cnt := 0;
   END_IF;
   #_w3 := "reset" AND NOT "抢答器LAD数据块_1".cache[9];   // rising edge of "reset"
   "抢答器LAD数据块_1".cache[9] := "reset";
   IF #_w3 THEN
       "抢答器LAD数据块_1".success_a := FALSE;
       "抢答器LAD数据块_1".success_b := FALSE;
       "抢答器LAD数据块_1".success_c := FALSE;
       "抢答器LAD数据块_1".success_d := FALSE;
       "抢答器LAD数据块_1".started := FALSE;
       "抢答器LAD数据块_1".success := FALSE;
       "light_a" := FALSE;
       "light_b" := FALSE;
       "light_c" := FALSE;
       "light_d" := FALSE;
   END_IF;
END_REGION

REGION Network 3
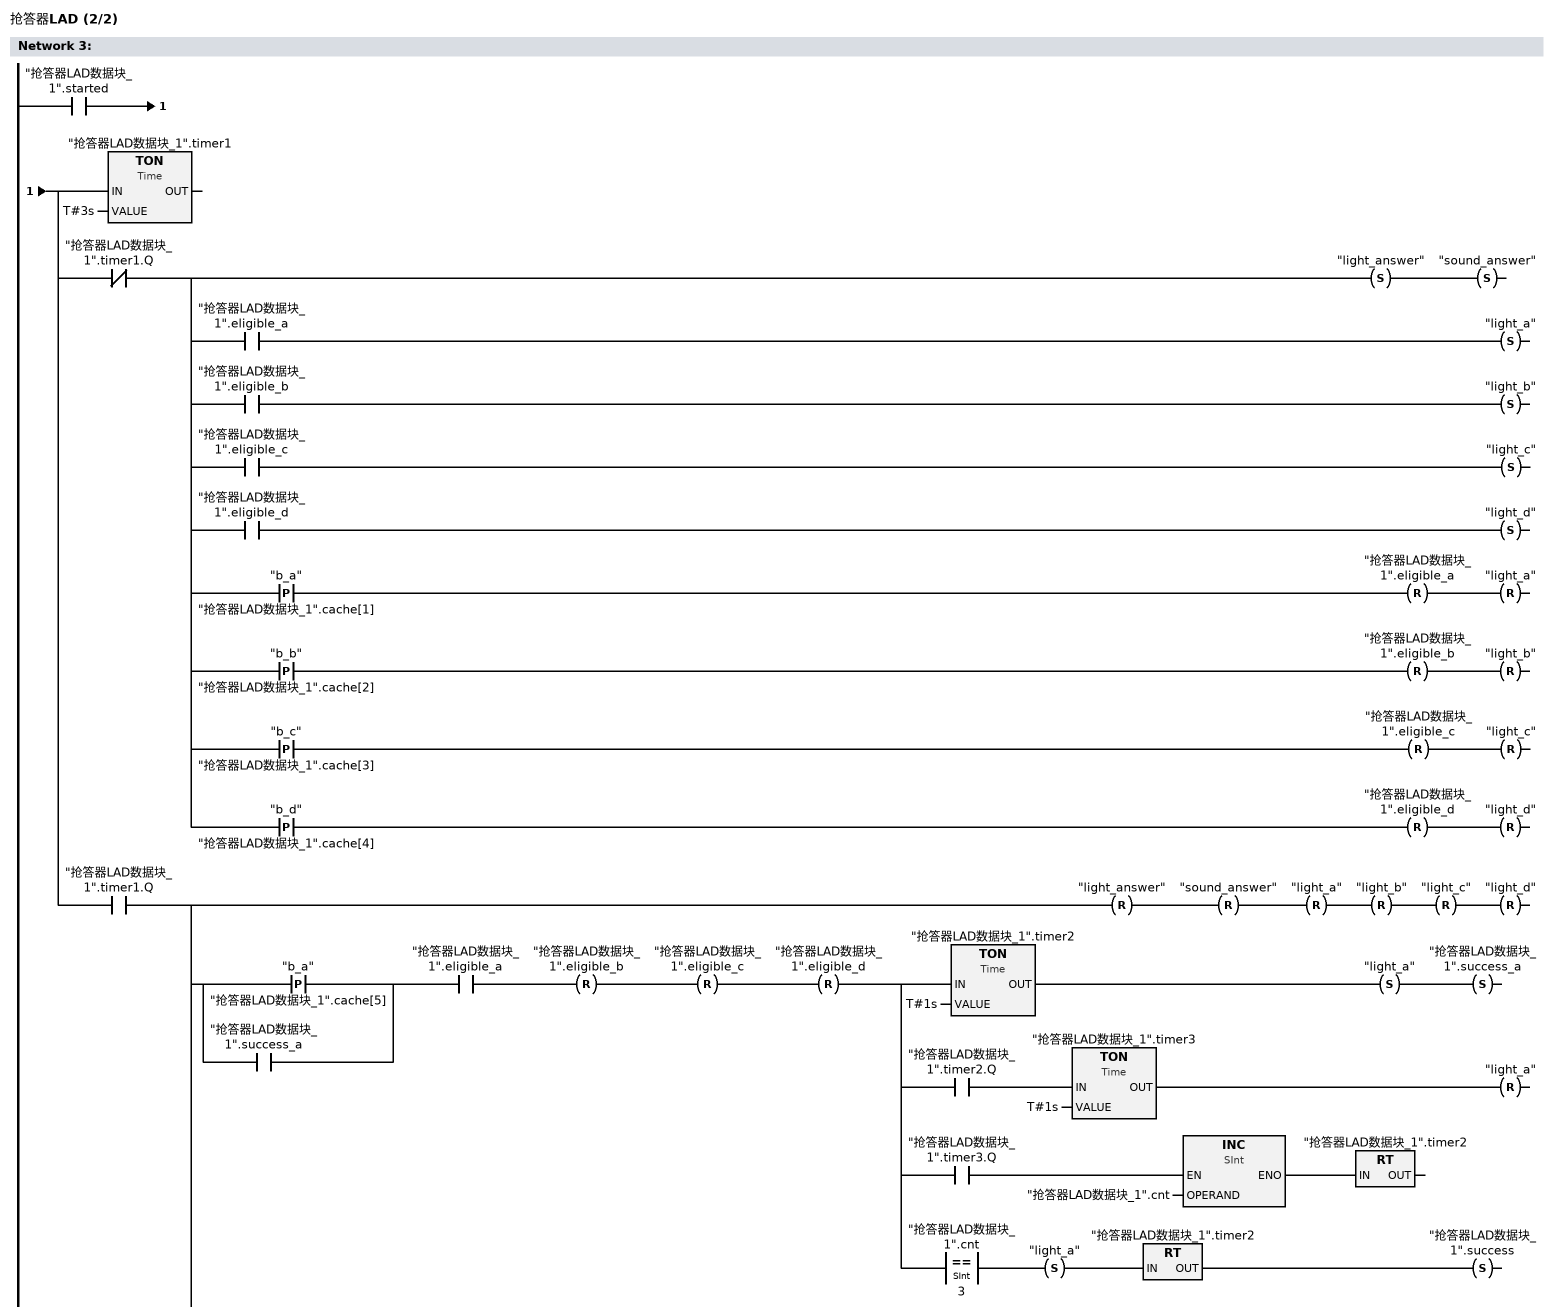
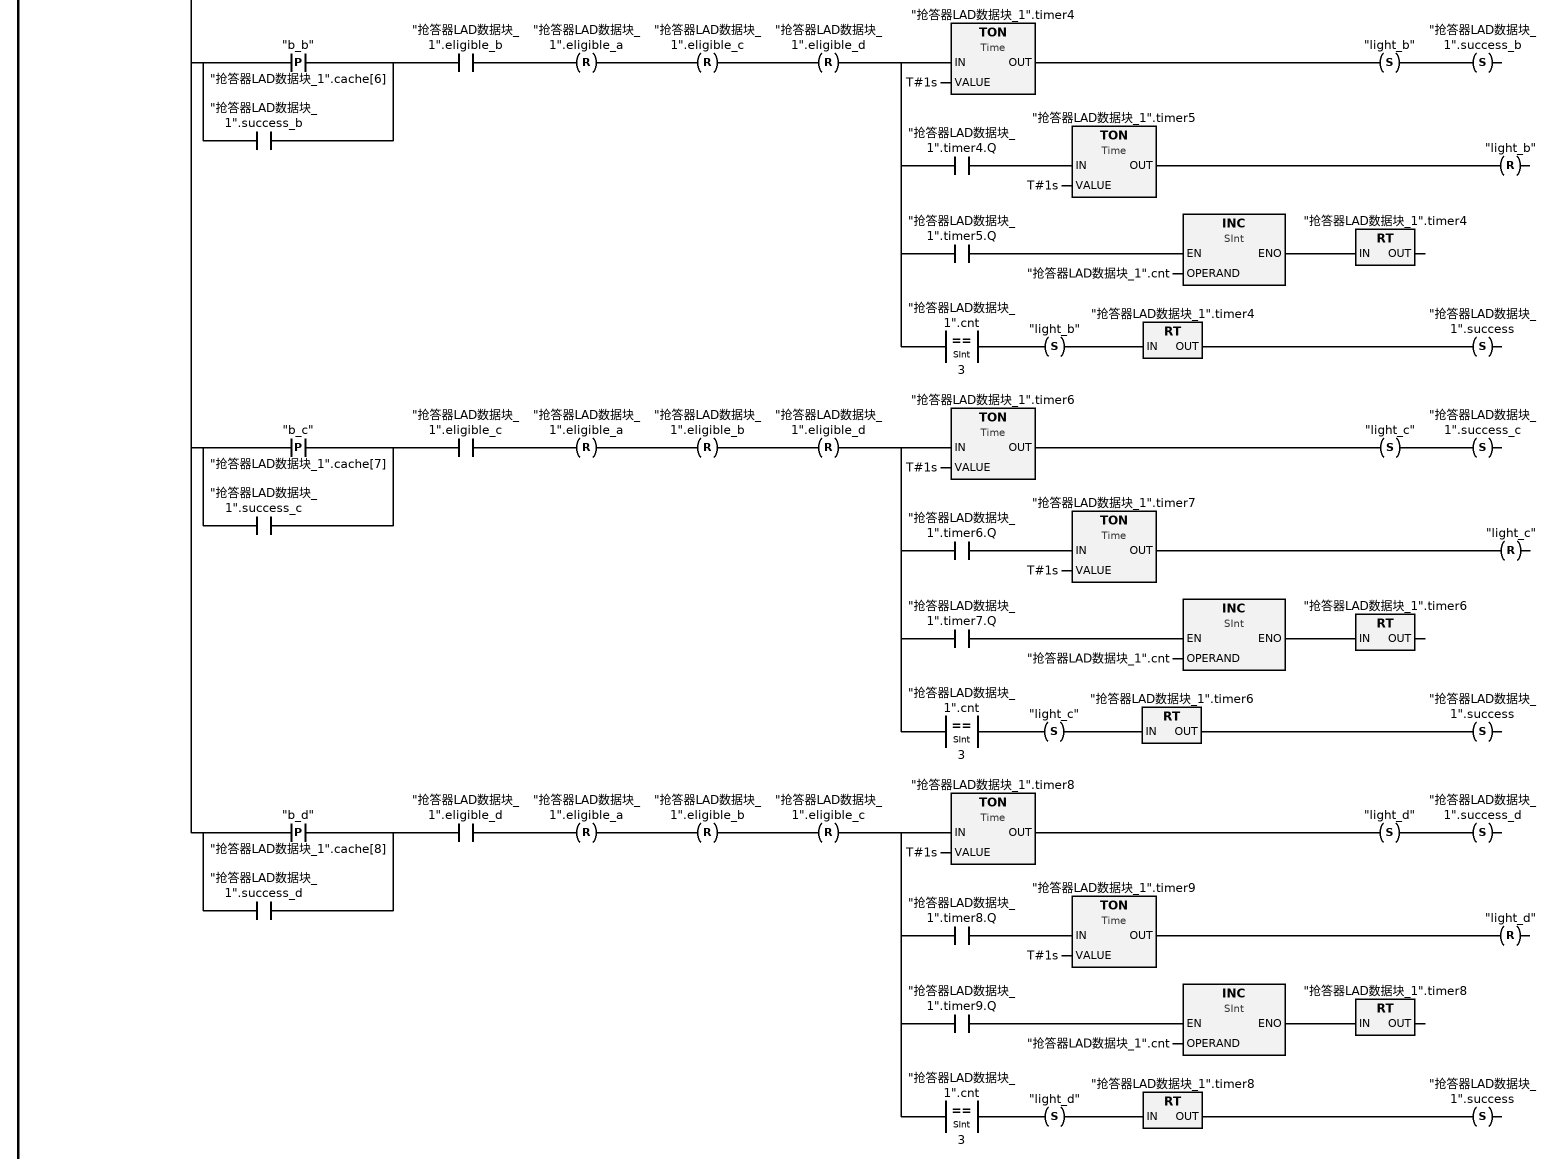
   "抢答器LAD数据块_1".timer1.TON(IN := "抢答器LAD数据块_1".started, PT := T#3s);   // TON coil
   #_w1 := "抢答器LAD数据块_1".started AND NOT "抢答器LAD数据块_1".timer1.Q;
   IF #_w1 THEN
       "light_answer" := TRUE;
       "sound_answer" := TRUE;
   END_IF;
   IF #_w1 AND "抢答器LAD数据块_1".eligible_a THEN "light_a" := TRUE; END_IF;
   IF #_w1 AND "抢答器LAD数据块_1".eligible_b THEN "light_b" := TRUE; END_IF;
   IF #_w1 AND "抢答器LAD数据块_1".eligible_c THEN "light_c" := TRUE; END_IF;
   IF #_w1 AND "抢答器LAD数据块_1".eligible_d THEN "light_d" := TRUE; END_IF;
   #_w2 := #_w1 AND "b_a" AND NOT "抢答器LAD数据块_1".cache[1];   // rising edge of "b_a"
   "抢答器LAD数据块_1".cache[1] := "b_a";
   IF #_w2 THEN
       "抢答器LAD数据块_1".eligible_a := FALSE;
       "light_a" := FALSE;
   END_IF;
   #_w3 := #_w1 AND "b_b" AND NOT "抢答器LAD数据块_1".cache[2];   // rising edge of "b_b"
   "抢答器LAD数据块_1".cache[2] := "b_b";
   IF #_w3 THEN
       "抢答器LAD数据块_1".eligible_b := FALSE;
       "light_b" := FALSE;
   END_IF;
   #_w4 := #_w1 AND "b_c" AND NOT "抢答器LAD数据块_1".cache[3];   // rising edge of "b_c"
   "抢答器LAD数据块_1".cache[3] := "b_c";
   IF #_w4 THEN
       "抢答器LAD数据块_1".eligible_c := FALSE;
       "light_c" := FALSE;
   END_IF;
   #_w5 := #_w1 AND "b_d" AND NOT "抢答器LAD数据块_1".cache[4];   // rising edge of "b_d"
   "抢答器LAD数据块_1".cache[4] := "b_d";
   IF #_w5 THEN
       "抢答器LAD数据块_1".eligible_d := FALSE;
       "light_d" := FALSE;
   END_IF;
   #_w6 := "抢答器LAD数据块_1".started AND "抢答器LAD数据块_1".timer1.Q;
   IF #_w6 THEN
       "light_answer" := FALSE;
       "sound_answer" := FALSE;
       "light_a" := FALSE;
       "light_b" := FALSE;
       "light_c" := FALSE;
       "light_d" := FALSE;
   END_IF;
   #_w7 := #_w6 AND "b_a" AND NOT "抢答器LAD数据块_1".cache[5];   // rising edge of "b_a"
   "抢答器LAD数据块_1".cache[5] := "b_a";
   #_w8 := (#_w7 OR (#_w6 AND "抢答器LAD数据块_1".success_a)) AND "抢答器LAD数据块_1".eligible_a;
   IF #_w8 THEN
       "抢答器LAD数据块_1".eligible_b := FALSE;
       "抢答器LAD数据块_1".eligible_c := FALSE;
       "抢答器LAD数据块_1".eligible_d := FALSE;
   END_IF;
   "抢答器LAD数据块_1".timer2.TON(IN := #_w8, PT := T#1s);   // TON coil
   IF #_w8 THEN
       "light_a" := TRUE;
       "抢答器LAD数据块_1".success_a := TRUE;
   END_IF;
   #_w9 := #_w8 AND "抢答器LAD数据块_1".timer2.Q;
   "抢答器LAD数据块_1".timer3.TON(IN := #_w9, PT := T#1s);   // TON coil
   IF #_w9 THEN "light_a" := FALSE; END_IF;
   #_w10 := #_w8 AND "抢答器LAD数据块_1".timer3.Q;
   IF #_w10 THEN
       "抢答器LAD数据块_1".cnt := "抢答器LAD数据块_1".cnt + 1;
       RESET_TIMER("抢答器LAD数据块_1".timer2);
   END_IF;
   #_w11 := #_w8 AND ("抢答器LAD数据块_1".cnt = 3);
   IF #_w11 THEN
       "light_a" := TRUE;
       RESET_TIMER("抢答器LAD数据块_1".timer2);
       "抢答器LAD数据块_1".success := TRUE;
   END_IF;
   #_w12 := #_w6 AND "b_b" AND NOT "抢答器LAD数据块_1".cache[6];   // rising edge of "b_b"
   "抢答器LAD数据块_1".cache[6] := "b_b";
   #_w13 := (#_w12 OR (#_w6 AND "抢答器LAD数据块_1".success_b)) AND "抢答器LAD数据块_1".eligible_b;
   IF #_w13 THEN
       "抢答器LAD数据块_1".eligible_a := FALSE;
       "抢答器LAD数据块_1".eligible_c := FALSE;
       "抢答器LAD数据块_1".eligible_d := FALSE;
   END_IF;
   "抢答器LAD数据块_1".timer4.TON(IN := #_w13, PT := T#1s);   // TON coil
   IF #_w13 THEN
       "light_b" := TRUE;
       "抢答器LAD数据块_1".success_b := TRUE;
   END_IF;
   #_w14 := #_w13 AND "抢答器LAD数据块_1".timer4.Q;
   "抢答器LAD数据块_1".timer5.TON(IN := #_w14, PT := T#1s);   // TON coil
   IF #_w14 THEN "light_b" := FALSE; END_IF;
   #_w15 := #_w13 AND "抢答器LAD数据块_1".timer5.Q;
   IF #_w15 THEN
       "抢答器LAD数据块_1".cnt := "抢答器LAD数据块_1".cnt + 1;
       RESET_TIMER("抢答器LAD数据块_1".timer4);
   END_IF;
   #_w16 := #_w13 AND ("抢答器LAD数据块_1".cnt = 3);
   IF #_w16 THEN
       "light_b" := TRUE;
       RESET_TIMER("抢答器LAD数据块_1".timer4);
       "抢答器LAD数据块_1".success := TRUE;
   END_IF;
   #_w17 := #_w6 AND "b_c" AND NOT "抢答器LAD数据块_1".cache[7];   // rising edge of "b_c"
   "抢答器LAD数据块_1".cache[7] := "b_c";
   #_w18 := (#_w17 OR (#_w6 AND "抢答器LAD数据块_1".success_c)) AND "抢答器LAD数据块_1".eligible_c;
   IF #_w18 THEN
       "抢答器LAD数据块_1".eligible_a := FALSE;
       "抢答器LAD数据块_1".eligible_b := FALSE;
       "抢答器LAD数据块_1".eligible_d := FALSE;
   END_IF;
   "抢答器LAD数据块_1".timer6.TON(IN := #_w18, PT := T#1s);   // TON coil
   IF #_w18 THEN
       "light_c" := TRUE;
       "抢答器LAD数据块_1".success_c := TRUE;
   END_IF;
   #_w19 := #_w18 AND "抢答器LAD数据块_1".timer6.Q;
   "抢答器LAD数据块_1".timer7.TON(IN := #_w19, PT := T#1s);   // TON coil
   IF #_w19 THEN "light_c" := FALSE; END_IF;
   #_w20 := #_w18 AND "抢答器LAD数据块_1".timer7.Q;
   IF #_w20 THEN
       "抢答器LAD数据块_1".cnt := "抢答器LAD数据块_1".cnt + 1;
       RESET_TIMER("抢答器LAD数据块_1".timer6);
   END_IF;
   #_w21 := #_w18 AND ("抢答器LAD数据块_1".cnt = 3);
   IF #_w21 THEN
       "light_c" := TRUE;
       RESET_TIMER("抢答器LAD数据块_1".timer6);
       "抢答器LAD数据块_1".success := TRUE;
   END_IF;
   #_w22 := #_w6 AND "b_d" AND NOT "抢答器LAD数据块_1".cache[8];   // rising edge of "b_d"
   "抢答器LAD数据块_1".cache[8] := "b_d";
   #_w23 := (#_w22 OR (#_w6 AND "抢答器LAD数据块_1".success_d)) AND "抢答器LAD数据块_1".eligible_d;
   IF #_w23 THEN
       "抢答器LAD数据块_1".eligible_a := FALSE;
       "抢答器LAD数据块_1".eligible_b := FALSE;
       "抢答器LAD数据块_1".eligible_c := FALSE;
   END_IF;
   "抢答器LAD数据块_1".timer8.TON(IN := #_w23, PT := T#1s);   // TON coil
   IF #_w23 THEN
       "light_d" := TRUE;
       "抢答器LAD数据块_1".success_d := TRUE;
   END_IF;
   #_w24 := #_w23 AND "抢答器LAD数据块_1".timer8.Q;
   "抢答器LAD数据块_1".timer9.TON(IN := #_w24, PT := T#1s);   // TON coil
   IF #_w24 THEN "light_d" := FALSE; END_IF;
   #_w25 := #_w23 AND "抢答器LAD数据块_1".timer9.Q;
   IF #_w25 THEN
       "抢答器LAD数据块_1".cnt := "抢答器LAD数据块_1".cnt + 1;
       RESET_TIMER("抢答器LAD数据块_1".timer8);
   END_IF;
   #_w26 := #_w23 AND ("抢答器LAD数据块_1".cnt = 3);
   IF #_w26 THEN
       "light_d" := TRUE;
       RESET_TIMER("抢答器LAD数据块_1".timer8);
       "抢答器LAD数据块_1".success := TRUE;
   END_IF;
END_REGION
END_FUNCTION